TYPE ST_System_WT_HWW_Steuerung :
STRUCT
	Freigabe				: ST_Steuerung_auto_manu_BOOL;
	Freigabe_Deakt		: ST_Steuerung_auto_manu_BOOL;
	Betrieb_Anford		: ST_Steuerung_auto_manu_opti_BOOL;

	Regelung_Sollw		: ST_Steuerung_auto_manu_opti_REAL;

	Quittierung			: BOOL;
END_STRUCT
END_TYPE

(* stored: Version 1.1.0.1, ProductVersion 3.1.4024.9
   DUT ST_System_WT_HWW_Steuerung: Id {8b8353bd-f6b8-46ae-b4eb-de11362f1880} *)
